LIN {X 0,Y 101.86,Z 670.766,A -85,B 0,C 180,E1 -28292.306,E2 -28292.306} C_VEL
LIN {X 0,Y 95.188,Z 678.477,A -85,B 0,C 180,E1 -28295.693,E2 -28295.693} C_VEL
LIN {X 0,Y 87.721,Z 685.98,A -85,B 0,C 180,E1 -28300.438,E2 -28300.438} C_VEL
LIN {X 0,Y 80.748,Z 692,A -85,B 0,C 180,E1 -28305.87,E2 -28305.87} C_VEL
LIN {X 0,Y 74.603,Z 696.757,A -85,B 0,C 180,E1 -28312.242,E2 -28312.242} C_VEL
LIN {X 0,Y 69.596,Z 700.393,A -85,B 0,C 180,E1 -28319.675,E2 -28319.675} C_VEL
LIN {X 0,Y 66.959,Z 702.265,A -85,B 0,C 180,E1 -28325.176,E2 -28325.176} C_VEL
LIN {X 0,Y 64.891,Z 703.687,A -85,B 0,C 180,E1 -28331.04,E2 -28331.04} C_VEL
LIN {X 0,Y 63.469,Z 704.685,A -85,B 0,C 180,E1 -28337.206,E2 -28337.206} C_VEL
LIN {X 0,Y 62.687,Z 705.298,A -85,B 0,C 180,E1 -28343.564,E2 -28343.564} C_VEL
LIN {X 0,Y 62.554,Z 705.526,A -85,B 0,C 180,E1 -28350.001,E2 -28350.001} C_VEL
LIN {X 0,Y 62.682,Z 705.324,A -85,B 0,C 180,E1 -28356.439,E2 -28356.439} C_VEL
LIN {X 0,Y 63.445,Z 704.728,A -85,B 0,C 180,E1 -28362.801,E2 -28362.801} C_VEL
LIN {X 0,Y 64.821,Z 703.747,A -85,B 0,C 180,E1 -28368.983,E2 -28368.983} C_VEL
LIN {X 0,Y 66.882,Z 702.358,A -85,B 0,C 180,E1 -28374.856,E2 -28374.856} C_VEL
LIN {X 0,Y 71.032,Z 699.448,A -85,B 0,C 180,E1 -28382.97,E2 -28382.97} C_VEL
LIN {X 0,Y 76.493,Z 695.492,A -85,B 0,C 180,E1 -28390.028,E2 -28390.028} C_VEL
LIN {X 0,Y 82.906,Z 690.364,A -85,B 0,C 180,E1 -28396.102,E2 -28396.102} C_VEL
LIN {X 0,Y 90.621,Z 683.358,A -85,B 0,C 180,E1 -28401.652,E2 -28401.652} C_VEL
LIN {X 0,Y 97.748,Z 675.871,A -85,B 0,C 180,E1 -28405.777,E2 -28405.777} C_VEL
LIN {X 0,Y 104.595,Z 667.648,A -85,B 0,C 180,E1 -28408.95,E2 -28408.95} C_VEL
LIN {X 0,Y 111.753,Z 657.491,A -85,B 0,C 180,E1 -28411.697,E2 -28411.697} C_VEL
LIN {X 0,Y 118.381,Z 646.062,A -85,B 0,C 180,E1 -28413.89,E2 -28413.89} C_VEL
LIN {X 0,Y 123.615,Z 634.711,A -85,B 0,C 180,E1 -28415.461,E2 -28415.461} C_VEL
LIN {X 0,Y 128.197,Z 621.782,A -85,B 0,C 180,E1 -28416.675,E2 -28416.675} C_VEL
LIN {X 0,Y 131.423,Z 608.945,A -85,B 0,C 180,E1 -28417.489,E2 -28417.489} C_VEL
LIN {X 0,Y 133.473,Z 595.213,A -85,B 0,C 180,E1 -28418.011,E2 -28418.011} C_VEL
LIN {X 0,Y 138.268,Z 548.092,A -85,B 0,C 180,E1 -28419.546,E2 -28419.546} C_VEL
LIN {X 0,Y 138.309,Z 545.503,A -85,B 0,C 180,E1 -28419.878,E2 -28419.878} C_VEL
LIN {X 0,Y 136.481,Z 538.988,A -85,B 0,C 180,E1 -28423.201,E2 -28423.201} C_VEL
LIN {X 0,Y 135.049,Z 534.594,A -85,B 0,C 180,E1 -28426.265,E2 -28426.265} C_VEL
LIN {X 0,Y 134.032,Z 531.605,A -85,B 0,C 180,E1 -28428.947,E2 -28428.947} C_VEL
LIN {X 0,Y 132.897,Z 528.182,A -85,B 0,C 180,E1 -28433.166,E2 -28433.166} C_VEL
LIN {X 0,Y 132.282,Z 525.748,A -85,B 0,C 180,E1 -28438.478,E2 -28438.478} C_VEL
LIN {X 0,Y 132.299,Z 525.196,A -85,B 0,C 180,E1 -28440,E2 -28440} C_VEL
LIN {X 0,Y 132.523,Z 525.208,A -85,B 0,C 180,E1 -28443.42,E2 -28443.42} C_VEL
LIN {X 0,Y 133.793,Z 527.549,A -85,B 0,C 180,E1 -28449.448,E2 -28449.448} C_VEL
LIN {X 0,Y 135.294,Z 530.109,A -85,B 0,C 180,E1 -28453.327,E2 -28453.327} C_VEL
LIN {X 0,Y 137.511,Z 534.497,A -85,B 0,C 180,E1 -28457.569,E2 -28457.569} C_VEL
LIN {X 0,Y 138.613,Z 536.926,A -85,B 0,C 180,E1 -28459.339,E2 -28459.339} C_VEL
LIN {X 0,Y 137.874,Z 550.601,A -85,B 0,C 180,E1 -28460.537,E2 -28460.537} C_VEL
LIN {X 0,Y 132.225,Z 603.924,A -85,B 0,C 180,E1 -28462.263,E2 -28462.263} C_VEL
LIN {X 0,Y 129.662,Z 616.387,A -85,B 0,C 180,E1 -28462.86,E2 -28462.86} C_VEL
LIN {X 0,Y 125.786,Z 629.073,A -85,B 0,C 180,E1 -28463.805,E2 -28463.805} C_VEL
LIN {X 0,Y 121.232,Z 640.398,A -85,B 0,C 180,E1 -28465.066,E2 -28465.066} C_VEL
LIN {X 0,Y 115.246,Z 652.046,A -85,B 0,C 180,E1 -28466.889,E2 -28466.889} C_VEL
LIN {X 0,Y 108.673,Z 662.454,A -85,B 0,C 180,E1 -28469.182,E2 -28469.182} C_VEL
LIN {X 0,Y 101.589,Z 671.843,A -85,B 0,C 180,E1 -28472.062,E2 -28472.062} C_VEL
LIN {X 0,Y 93.505,Z 680.856,A -85,B 0,C 180,E1 -28476.099,E2 -28476.099} C_VEL
LIN {X 0,Y 85.896,Z 688.299,A -85,B 0,C 180,E1 -28481.118,E2 -28481.118} C_VEL
LIN {X 0,Y 80.359,Z 693.02,A -85,B 0,C 180,E1 -28485.599,E2 -28485.599} C_VEL
LIN {X 0,Y 74.261,Z 697.769,A -85,B 0,C 180,E1 -28492.036,E2 -28492.036} C_VEL
LIN {X 0,Y 69.197,Z 701.394,A -85,B 0,C 180,E1 -28499.48,E2 -28499.48} C_VEL
LIN {X 0,Y 66.631,Z 703.263,A -85,B 0,C 180,E1 -28505.044,E2 -28505.044} C_VEL
LIN {X 0,Y 64.645,Z 704.669,A -85,B 0,C 180,E1 -28510.964,E2 -28510.964} C_VEL
LIN {X 0,Y 63.349,Z 705.663,A -85,B 0,C 180,E1 -28517.179,E2 -28517.179} C_VEL
LIN {X 0,Y 62.666,Z 706.269,A -85,B 0,C 180,E1 -28523.56,E2 -28523.56} C_VEL
LIN {X 0,Y 62.617,Z 706.48,A -85,B 0,C 180,E1 -28529.999,E2 -28529.999} C_VEL
LIN {X 0,Y 62.666,Z 706.25,A -85,B 0,C 180,E1 -28536.438,E2 -28536.438} C_VEL
LIN {X 0,Y 63.349,Z 705.631,A -85,B 0,C 180,E1 -28542.819,E2 -28542.819} C_VEL
LIN {X 0,Y 64.645,Z 704.625,A -85,B 0,C 180,E1 -28549.034,E2 -28549.034} C_VEL
LIN {X 0,Y 66.632,Z 703.194,A -85,B 0,C 180,E1 -28554.954,E2 -28554.954} C_VEL
LIN {X 0,Y 70.759,Z 700.231,A -85,B 0,C 180,E1 -28563.111,E2 -28563.111} C_VEL
LIN {X 0,Y 76.222,Z 696.212,A -85,B 0,C 180,E1 -28570.197,E2 -28570.197} C_VEL
LIN {X 0,Y 82.628,Z 691.019,A -85,B 0,C 180,E1 -28576.3,E2 -28576.3} C_VEL
LIN {X 0,Y 89.725,Z 684.486,A -85,B 0,C 180,E1 -28581.561,E2 -28581.561} C_VEL
LIN {X 0,Y 97.461,Z 676.359,A -85,B 0,C 180,E1 -28586.023,E2 -28586.023} C_VEL
LIN {X 0,Y 104.564,Z 667.747,A -85,B 0,C 180,E1 -28589.248,E2 -28589.248} C_VEL
LIN {X 0,Y 104.524,Z 666.501,A -85,B 0,C 180,E1 -28590.516,E2 -28590.516} C_VEL
LIN {X 0,Y 98.912,Z 662.815,A -85,B 0,C 180,E1 -28602.135,E2 -28602.135} C_VEL
LIN {X 0,Y 98.359,Z 659.574,A -85,B 0,C 180,E1 -28609.71,E2 -28609.71} C_VEL
LIN {X 0,Y 99.161,Z 657.199,A -85,B 0,C 180,E1 -28613.724,E2 -28613.724} C_VEL
LIN {X 0,Y 99.935,Z 655.554,A -85,B 0,C 180,E1 -28616.976,E2 -28616.976} C_VEL
LIN {X 0,Y 102.399,Z 652.842,A -85,B 0,C 180,E1 -28626.921,E2 -28626.921} C_VEL
LIN {X 0,Y 104.174,Z 651.421,A -85,B 0,C 180,E1 -28629.967,E2 -28629.967} C_VEL
LIN {X 0,Y 104.937,Z 650.77,A -85,B 0,C 180,E1 -28630.903,E2 -28630.903} C_VEL
LIN {X 0,Y 109.265,Z 646.893,A -85,B 0,C 180,E1 -28635.098,E2 -28635.098} C_VEL
LIN {X 0,Y 116.042,Z 640.504,A -85,B 0,C 180,E1 -28639.805,E2 -28639.805} C_VEL
LIN {X 0,Y 119.153,Z 637.397,A -85,B 0,C 180,E1 -28641.632,E2 -28641.632} C_VEL
LIN {X 0,Y 118.879,Z 638.512,A -85,B 0,C 180,E1 -28642.044,E2 -28642.044} C_VEL
LIN {X 0,Y 113.178,Z 649.684,A -85,B 0,C 180,E1 -28643.662,E2 -28643.662} C_VEL
LIN {X 0,Y 106.362,Z 660.356,A -85,B 0,C 180,E1 -28645.805,E2 -28645.805} C_VEL
LIN {X 0,Y 98.252,Z 670.818,A -85,B 0,C 180,E1 -28648.808,E2 -28648.808} C_VEL
LIN {X 0,Y 91.212,Z 678.529,A -85,B 0,C 180,E1 -28652.053,E2 -28652.053} C_VEL
LIN {X 0,Y 83.223,Z 686.089,A -85,B 0,C 180,E1 -28656.757,E2 -28656.757} C_VEL
LIN {X 0,Y 75.792,Z 692.054,A -85,B 0,C 180,E1 -28662.114,E2 -28662.114} C_VEL
LIN {X 0,Y 69.122,Z 696.812,A -85,B 0,C 180,E1 -28668.633,E2 -28668.633} C_VEL
LIN {X 0,Y 63.538,Z 700.448,A -85,B 0,C 180,E1 -28676.424,E2 -28676.424} C_VEL
LIN {X 0,Y 60.561,Z 702.319,A -85,B 0,C 180,E1 -28682.343,E2 -28682.343} C_VEL
LIN {X 0,Y 58.212,Z 703.741,A -85,B 0,C 180,E1 -28688.766,E2 -28688.766} C_VEL
LIN {X 0,Y 55.63,Z 705.352,A -85,B 0,C 180,E1 -28702.743,E2 -28702.743} C_VEL
LIN {X 0,Y 55.473,Z 705.58,A -85,B 0,C 180,E1 -28710.001,E2 -28710.001} C_VEL
LIN {X 0,Y 55.626,Z 705.378,A -85,B 0,C 180,E1 -28717.259,E2 -28717.259} C_VEL
LIN {X 0,Y 56.529,Z 704.781,A -85,B 0,C 180,E1 -28724.399,E2 -28724.399} C_VEL
LIN {X 0,Y 58.15,Z 703.8,A -85,B 0,C 180,E1 -28731.26,E2 -28731.26} C_VEL
LIN {X 0,Y 60.49,Z 702.411,A -85,B 0,C 180,E1 -28737.695,E2 -28737.695} C_VEL
LIN {X 0,Y 65.174,Z 699.501,A -85,B 0,C 180,E1 -28746.378,E2 -28746.378} C_VEL
LIN {X 0,Y 71.197,Z 695.544,A -85,B 0,C 180,E1 -28753.709,E2 -28753.709} C_VEL
LIN {X 0,Y 78.142,Z 690.415,A -85,B 0,C 180,E1 -28759.862,E2 -28759.862} C_VEL
LIN {X 0,Y 85.789,Z 683.952,A -85,B 0,C 180,E1 -28765.008,E2 -28765.008} C_VEL
LIN {X 0,Y 93.93,Z 675.919,A -85,B 0,C 180,E1 -28769.368,E2 -28769.368} C_VEL
LIN {X 0,Y 101.109,Z 667.693,A -85,B 0,C 180,E1 -28772.407,E2 -28772.407} C_VEL
LIN {X 0,Y 108.564,Z 657.532,A -85,B 0,C 180,E1 -28775.001,E2 -28775.001} C_VEL
LIN {X 0,Y 115.434,Z 646.099,A -85,B 0,C 180,E1 -28777.054,E2 -28777.054} C_VEL
LIN {X 0,Y 120.841,Z 634.739,A -85,B 0,C 180,E1 -28778.522,E2 -28778.522} C_VEL
LIN {X 0,Y 125.558,Z 621.799,A -85,B 0,C 180,E1 -28779.649,E2 -28779.649} C_VEL
LIN {X 0,Y 128.829,Z 609.172,A -85,B 0,C 180,E1 -28780.39,E2 -28780.39} C_VEL
LIN {X 0,Y 130.949,Z 595.406,A -85,B 0,C 180,E1 -28780.886,E2 -28780.886} C_VEL
LIN {X 0,Y 135.81,Z 549.367,A -85,B 0,C 180,E1 -28782.304,E2 -28782.304} C_VEL
LIN {X 0,Y 134.47,Z 544.016,A -85,B 0,C 180,E1 -28785.239,E2 -28785.239} C_VEL
LIN {X 0,Y 132.962,Z 538.749,A -85,B 0,C 180,E1 -28789.339,E2 -28789.339} C_VEL
LIN {X 0,Y 131.864,Z 535.005,A -85,B 0,C 180,E1 -28793.881,E2 -28793.881} C_VEL
LIN {X 0,Y 131.402,Z 532.741,A -85,B 0,C 180,E1 -28798.851,E2 -28798.851} C_VEL
LIN {X 0,Y 131.424,Z 532.32,A -85,B 0,C 180,E1 -28800,E2 -28800} C_VEL
LIN {X 0,Y 131.67,Z 532.377,A -85,B 0,C 180,E1 -28803.634,E2 -28803.634} C_VEL
LIN {X 0,Y 132.86,Z 534.677,A -85,B 0,C 180,E1 -28809.323,E2 -28809.323} C_VEL
LIN {X 0,Y 134.08,Z 536.98,A -85,B 0,C 180,E1 -28812.679,E2 -28812.679} C_VEL
LIN {X 0,Y 135.868,Z 540.882,A -85,B 0,C 180,E1 -28816.432,E2 -28816.432} C_VEL
LIN {X 0,Y 136.117,Z 541.431,A -85,B 0,C 180,E1 -28816.884,E2 -28816.884} C_VEL
LIN {X 0,Y 135.492,Z 551.207,A -85,B 0,C 180,E1 -28817.742,E2 -28817.742} C_VEL
LIN {X 0,Y 129.707,Z 603.961,A -85,B 0,C 180,E1 -28819.366,E2 -28819.366} C_VEL
LIN {X 0,Y 126.879,Z 617.11,A -85,B 0,C 180,E1 -28819.96,E2 -28819.96} C_VEL
LIN {X 0,Y 122.703,Z 630.146,A -85,B 0,C 180,E1 -28820.879,E2 -28820.879} C_VEL
LIN {X 0,Y 117.624,Z 641.987,A -85,B 0,C 180,E1 -28822.159,E2 -28822.159} C_VEL
LIN {X 0,Y 111.461,Z 653.275,A -85,B 0,C 180,E1 -28823.895,E2 -28823.895} C_VEL
LIN {X 0,Y 104.642,Z 663.464,A -85,B 0,C 180,E1 -28826.063,E2 -28826.063} C_VEL
LIN {X 0,Y 97.991,Z 671.797,A -85,B 0,C 180,E1 -28828.526,E2 -28828.526} C_VEL
LIN {X 0,Y 89.498,Z 680.808,A -85,B 0,C 180,E1 -28832.416,E2 -28832.416} C_VEL
LIN {X 0,Y 82.031,Z 687.662,A -85,B 0,C 180,E1 -28836.85,E2 -28836.85} C_VEL
LIN {X 0,Y 75.449,Z 692.969,A -85,B 0,C 180,E1 -28841.823,E2 -28841.823} C_VEL
LIN {X 0,Y 68.79,Z 697.717,A -85,B 0,C 180,E1 -28848.387,E2 -28848.387} C_VEL
LIN {X 0,Y 63.157,Z 701.341,A -85,B 0,C 180,E1 -28856.192,E2 -28856.192} C_VEL
LIN {X 0,Y 60.238,Z 703.21,A -85,B 0,C 180,E1 -28862.18,E2 -28862.18} C_VEL
LIN {X 0,Y 57.959,Z 704.615,A -85,B 0,C 180,E1 -28868.667,E2 -28868.667} C_VEL
LIN {X 0,Y 56.418,Z 705.609,A -85,B 0,C 180,E1 -28875.572,E2 -28875.572} C_VEL
LIN {X 0,Y 55.608,Z 706.215,A -85,B 0,C 180,E1 -28882.738,E2 -28882.738} C_VEL
LIN {X 0,Y 55.518,Z 706.426,A -85,B 0,C 180,E1 -28889.999,E2 -28889.999} C_VEL
LIN {X 0,Y 55.608,Z 706.196,A -85,B 0,C 180,E1 -28897.26,E2 -28897.26} C_VEL
LIN {X 0,Y 56.44,Z 705.577,A -85,B 0,C 180,E1 -28904.42,E2 -28904.42} C_VEL
LIN {X 0,Y 57.959,Z 704.57,A -85,B 0,C 180,E1 -28911.331,E2 -28911.331} C_VEL
LIN {X 0,Y 60.24,Z 703.139,A -85,B 0,C 180,E1 -28917.817,E2 -28917.817} C_VEL
LIN {X 0,Y 64.909,Z 700.176,A -85,B 0,C 180,E1 -28926.548,E2 -28926.548} C_VEL
LIN {X 0,Y 70.917,Z 696.158,A -85,B 0,C 180,E1 -28933.924,E2 -28933.924} C_VEL
LIN {X 0,Y 77.887,Z 690.966,A -85,B 0,C 180,E1 -28940.083,E2 -28940.083} C_VEL
LIN {X 0,Y 85.468,Z 684.432,A -85,B 0,C 180,E1 -28945.315,E2 -28945.315} C_VEL
LIN {X 0,Y 93.674,Z 676.307,A -85,B 0,C 180,E1 -28949.632,E2 -28949.632} C_VEL
LIN {X 0,Y 98.134,Z 671.326,A -85,B 0,C 180,E1 -28951.527,E2 -28951.527} C_VEL
LIN {X 0,Y 97.705,Z 670.632,A -85,B 0,C 180,E1 -28952.853,E2 -28952.853} C_VEL
LIN {X 0,Y 93.931,Z 667.818,A -85,B 0,C 180,E1 -28962.586,E2 -28962.586} C_VEL
LIN {X 0,Y 93.807,Z 664.313,A -85,B 0,C 180,E1 -28971.383,E2 -28971.383} C_VEL
LIN {X 0,Y 97.057,Z 659.101,A -85,B 0,C 180,E1 -28980,E2 -28980} C_VEL
LIN {X 0,Y 101.182,Z 654.304,A -85,B 0,C 180,E1 -28985.981,E2 -28985.981} C_VEL
LIN {X 0,Y 104.937,Z 650.77,A -85,B 0,C 180,E1 -28990.903,E2 -28990.903} C_VEL
LIN {X 0,Y 105.764,Z 650.311,A -85,B 0,C 180,E1 -28992.232,E2 -28992.232} C_VEL
LIN {X 0,Y 106.24,Z 650.817,A -85,B 0,C 180,E1 -28994.121,E2 -28994.121} C_VEL
LIN {X 0,Y 106.094,Z 652.648,A -85,B 0,C 180,E1 -28996.445,E2 -28996.445} C_VEL
LIN {X 0,Y 104.964,Z 656.019,A -85,B 0,C 180,E1 -28999.009,E2 -28999.009} C_VEL
LIN {X 0,Y 102.937,Z 660.296,A -85,B 0,C 180,E1 -29001.374,E2 -29001.374} C_VEL
LIN {X 0,Y 100.077,Z 664.814,A -85,B 0,C 180,E1 -29003.248,E2 -29003.248} C_VEL
LIN {X 0,Y 98.91,Z 666.324,A -85,B 0,C 180,E1 -29003.721,E2 -29003.721} C_VEL
LIN {X 0,Y 90.56,Z 675.661,A -85,B 0,C 180,E1 -29006.815,E2 -29006.815} C_VEL
LIN {X 0,Y 81.98,Z 683.754,A -85,B 0,C 180,E1 -29010.988,E2 -29010.988} C_VEL
LIN {X 0,Y 73.799,Z 690.26,A -85,B 0,C 180,E1 -29015.956,E2 -29015.956} C_VEL
LIN {X 0,Y 66.289,Z 695.43,A -85,B 0,C 180,E1 -29022.086,E2 -29022.086} C_VEL
LIN {X 0,Y 59.657,Z 699.429,A -85,B 0,C 180,E1 -29029.615,E2 -29029.615} C_VEL
LIN {X 0,Y 54.351,Z 702.374,A -85,B 0,C 180,E1 -29038.854,E2 -29038.854} C_VEL
LIN {X 0,Y 51.655,Z 703.796,A -85,B 0,C 180,E1 -29045.911,E2 -29045.911} C_VEL
LIN {X 0,Y 48.602,Z 705.406,A -85,B 0,C 180,E1 -29061.687,E2 -29061.687} C_VEL
LIN {X 0,Y 48.375,Z 705.634,A -85,B 0,C 180,E1 -29070.001,E2 -29070.001} C_VEL
LIN {X 0,Y 48.597,Z 705.431,A -85,B 0,C 180,E1 -29078.316,E2 -29078.316} C_VEL
LIN {X 0,Y 49.682,Z 704.835,A -85,B 0,C 180,E1 -29086.436,E2 -29086.436} C_VEL
LIN {X 0,Y 51.586,Z 703.854,A -85,B 0,C 180,E1 -29094.125,E2 -29094.125} C_VEL
LIN {X 0,Y 54.287,Z 702.465,A -85,B 0,C 180,E1 -29101.189,E2 -29101.189} C_VEL
LIN {X 0,Y 59.599,Z 699.553,A -85,B 0,C 180,E1 -29110.436,E2 -29110.436} C_VEL
LIN {X 0,Y 66.244,Z 695.595,A -85,B 0,C 180,E1 -29117.959,E2 -29117.959} C_VEL
LIN {X 0,Y 73.763,Z 690.465,A -85,B 0,C 180,E1 -29124.085,E2 -29124.085} C_VEL
LIN {X 0,Y 81.917,Z 684.001,A -85,B 0,C 180,E1 -29129.089,E2 -29129.089} C_VEL
LIN {X 0,Y 90.503,Z 675.966,A -85,B 0,C 180,E1 -29133.259,E2 -29133.259} C_VEL
LIN {X 0,Y 98.016,Z 667.739,A -85,B 0,C 180,E1 -29136.095,E2 -29136.095} C_VEL
LIN {X 0,Y 105.758,Z 657.574,A -85,B 0,C 180,E1 -29138.492,E2 -29138.492} C_VEL
LIN {X 0,Y 112.858,Z 646.135,A -85,B 0,C 180,E1 -29140.372,E2 -29140.372} C_VEL
LIN {X 0,Y 118.427,Z 634.767,A -85,B 0,C 180,E1 -29141.719,E2 -29141.719} C_VEL
LIN {X 0,Y 123.273,Z 621.816,A -85,B 0,C 180,E1 -29142.739,E2 -29142.739} C_VEL
LIN {X 0,Y 126.542,Z 609.541,A -85,B 0,C 180,E1 -29143.401,E2 -29143.401} C_VEL
LIN {X 0,Y 128.842,Z 595.013,A -85,B 0,C 180,E1 -29143.869,E2 -29143.869} C_VEL
LIN {X 0,Y 133.449,Z 552.752,A -85,B 0,C 180,E1 -29145.095,E2 -29145.095} C_VEL
LIN {X 0,Y 132.365,Z 548.001,A -85,B 0,C 180,E1 -29148.127,E2 -29148.127} C_VEL
LIN {X 0,Y 131.551,Z 544.776,A -85,B 0,C 180,E1 -29150.971,E2 -29150.971} C_VEL
LIN {X 0,Y 130.816,Z 541.688,A -85,B 0,C 180,E1 -29154.85,E2 -29154.85} C_VEL
LIN {X 0,Y 130.535,Z 539.591,A -85,B 0,C 180,E1 -29159.614,E2 -29159.614} C_VEL
LIN {X 0,Y 130.77,Z 539.401,A -85,B 0,C 180,E1 -29163.37,E2 -29163.37} C_VEL
LIN {X 0,Y 131.817,Z 541.585,A -85,B 0,C 180,E1 -29168.817,E2 -29168.817} C_VEL
LIN {X 0,Y 132.81,Z 543.717,A -85,B 0,C 180,E1 -29171.833,E2 -29171.833} C_VEL
LIN {X 0,Y 133.861,Z 546.095,A -85,B 0,C 180,E1 -29174.345,E2 -29174.345} C_VEL
LIN {X 0,Y 133.37,Z 552.487,A -85,B 0,C 180,E1 -29174.875,E2 -29174.875} C_VEL
LIN {X 0,Y 127.418,Z 604.64,A -85,B 0,C 180,E1 -29176.368,E2 -29176.368} C_VEL
LIN {X 0,Y 124.44,Z 617.833,A -85,B 0,C 180,E1 -29176.943,E2 -29176.943} C_VEL
LIN {X 0,Y 120.358,Z 630.122,A -85,B 0,C 180,E1 -29177.722,E2 -29177.722} C_VEL
LIN {X 0,Y 115.137,Z 641.953,A -85,B 0,C 180,E1 -29178.89,E2 -29178.89} C_VEL
LIN {X 0,Y 108.777,Z 653.236,A -85,B 0,C 180,E1 -29180.471,E2 -29180.471} C_VEL
LIN {X 0,Y 101.723,Z 663.42,A -85,B 0,C 180,E1 -29182.469,E2 -29182.469} C_VEL
LIN {X 0,Y 94.796,Z 671.751,A -85,B 0,C 180,E1 -29184.741,E2 -29184.741} C_VEL
LIN {X 0,Y 85.886,Z 680.76,A -85,B 0,C 180,E1 -29188.396,E2 -29188.396} C_VEL
LIN {X 0,Y 77.34,Z 688.121,A -85,B 0,C 180,E1 -29193.04,E2 -29193.04} C_VEL
LIN {X 0,Y 70.913,Z 692.918,A -85,B 0,C 180,E1 -29197.545,E2 -29197.545} C_VEL
LIN {X 0,Y 63.644,Z 697.665,A -85,B 0,C 180,E1 -29204.127,E2 -29204.127} C_VEL
LIN {X 0,Y 57.369,Z 701.288,A -85,B 0,C 180,E1 -29212.226,E2 -29212.226} C_VEL
LIN {X 0,Y 54.038,Z 703.157,A -85,B 0,C 180,E1 -29218.651,E2 -29218.651} C_VEL
LIN {X 0,Y 51.397,Z 704.561,A -85,B 0,C 180,E1 -29225.78,E2 -29225.78} C_VEL
LIN {X 0,Y 48.577,Z 706.161,A -85,B 0,C 180,E1 -29241.68,E2 -29241.68} C_VEL
LIN {X 0,Y 48.436,Z 706.372,A -85,B 0,C 180,E1 -29249.999,E2 -29249.999} C_VEL
LIN {X 0,Y 48.579,Z 706.141,A -85,B 0,C 180,E1 -29258.317,E2 -29258.317} C_VEL
LIN {X 0,Y 49.573,Z 705.522,A -85,B 0,C 180,E1 -29266.471,E2 -29266.471} C_VEL
LIN {X 0,Y 51.397,Z 704.516,A -85,B 0,C 180,E1 -29274.217,E2 -29274.217} C_VEL
LIN {X 0,Y 54.04,Z 703.084,A -85,B 0,C 180,E1 -29281.345,E2 -29281.345} C_VEL
LIN {X 0,Y 59.341,Z 700.122,A -85,B 0,C 180,E1 -29290.646,E2 -29290.646} C_VEL
LIN {X 0,Y 65.96,Z 696.104,A -85,B 0,C 180,E1 -29298.231,E2 -29298.231} C_VEL
LIN {X 0,Y 73.516,Z 690.912,A -85,B 0,C 180,E1 -29304.348,E2 -29304.348} C_VEL
LIN {X 0,Y 81.621,Z 684.379,A -85,B 0,C 180,E1 -29309.435,E2 -29309.435} C_VEL
LIN {X 0,Y 90.286,Z 676.255,A -85,B 0,C 180,E1 -29313.531,E2 -29313.531} C_VEL
LIN {X 0,Y 91.323,Z 674.766,A -85,B 0,C 180,E1 -29314.607,E2 -29314.607} C_VEL
LIN {X 0,Y 88.963,Z 672.945,A -85,B 0,C 180,E1 -29321.579,E2 -29321.579} C_VEL
LIN {X 0,Y 88.686,Z 669.789,A -85,B 0,C 180,E1 -29330.881,E2 -29330.881} C_VEL
LIN {X 0,Y 89.847,Z 667.724,A -85,B 0,C 180,E1 -29335.514,E2 -29335.514} C_VEL
LIN {X 0,Y 93.347,Z 663.616,A -85,B 0,C 180,E1 -29342.422,E2 -29342.422} C_VEL
LIN {X 0,Y 97.915,Z 659.201,A -85,B 0,C 180,E1 -29348.254,E2 -29348.254} C_VEL
LIN {X 0,Y 104.701,Z 653.863,A -85,B 0,C 180,E1 -29355.575,E2 -29355.575} C_VEL
LIN {X 0,Y 110.24,Z 649.405,A -85,B 0,C 180,E1 -29359.567,E2 -29359.567} C_VEL
LIN {X 0,Y 109.931,Z 650.703,A -85,B 0,C 180,E1 -29360.443,E2 -29360.443} C_VEL
LIN {X 0,Y 102.69,Z 661.452,A -85,B 0,C 180,E1 -29362.494,E2 -29362.494} C_VEL
LIN {X 0,Y 98.91,Z 666.324,A -85,B 0,C 180,E1 -29363.721,E2 -29363.721} C_VEL
LIN {X 0,Y 95.093,Z 670.569,A -85,B 0,C 180,E1 -29364.625,E2 -29364.625} C_VEL
LIN {X 0,Y 87.709,Z 677.086,A -85,B 0,C 180,E1 -29365.376,E2 -29365.376} C_VEL
LIN {X 0,Y 79.911,Z 682.975,A -85,B 0,C 180,E1 -29366.473,E2 -29366.473} C_VEL
LIN {X 0,Y 75.514,Z 686.232,A -85,B 0,C 180,E1 -29368.092,E2 -29368.092} C_VEL
LIN {X 0,Y 67.07,Z 692.161,A -85,B 0,C 180,E1 -29373.042,E2 -29373.042} C_VEL
LIN {X 0,Y 59.211,Z 696.92,A -85,B 0,C 180,E1 -29379.511,E2 -29379.511} C_VEL
LIN {X 0,Y 52.251,Z 700.557,A -85,B 0,C 180,E1 -29387.739,E2 -29387.739} C_VEL
LIN {X 0,Y 48.399,Z 702.428,A -85,B 0,C 180,E1 -29394.492,E2 -29394.492} C_VEL
LIN {X 0,Y 45.242,Z 703.85,A -85,B 0,C 180,E1 -29402.225,E2 -29402.225} C_VEL
LIN {X 0,Y 41.586,Z 705.461,A -85,B 0,C 180,E1 -29420.272,E2 -29420.272} C_VEL
LIN {X 0,Y 41.293,Z 705.688,A -85,B 0,C 180,E1 -29430.001,E2 -29430.001} C_VEL
LIN {X 0,Y 41.581,Z 705.485,A -85,B 0,C 180,E1 -29439.732,E2 -29439.732} C_VEL
LIN {X 0,Y 42.903,Z 704.889,A -85,B 0,C 180,E1 -29449.126,E2 -29449.126} C_VEL
LIN {X 0,Y 45.182,Z 703.907,A -85,B 0,C 180,E1 -29457.818,E2 -29457.818} C_VEL
LIN {X 0,Y 48.342,Z 702.518,A -85,B 0,C 180,E1 -29465.559,E2 -29465.559} C_VEL
LIN {X 0,Y 54.387,Z 699.606,A -85,B 0,C 180,E1 -29475.295,E2 -29475.295} C_VEL
LIN {X 0,Y 61.715,Z 695.647,A -85,B 0,C 180,E1 -29482.861,E2 -29482.861} C_VEL
LIN {X 0,Y 69.835,Z 690.516,A -85,B 0,C 180,E1 -29488.808,E2 -29488.808} C_VEL
LIN {X 0,Y 78.503,Z 684.05,A -85,B 0,C 180,E1 -29493.543,E2 -29493.543} C_VEL
LIN {X 0,Y 87.535,Z 676.014,A -85,B 0,C 180,E1 -29497.417,E2 -29497.417} C_VEL
LIN {X 0,Y 95.358,Z 667.784,A -85,B 0,C 180,E1 -29500.002,E2 -29500.002} C_VEL
LIN {X 0,Y 103.365,Z 657.615,A -85,B 0,C 180,E1 -29502.157,E2 -29502.157} C_VEL
LIN {X 0,Y 110.677,Z 646.172,A -85,B 0,C 180,E1 -29503.833,E2 -29503.833} C_VEL
LIN {X 0,Y 116.399,Z 634.795,A -85,B 0,C 180,E1 -29505.033,E2 -29505.033} C_VEL
LIN {X 0,Y 121.361,Z 621.831,A -85,B 0,C 180,E1 -29505.93,E2 -29505.93} C_VEL
LIN {X 0,Y 124.869,Z 608.767,A -85,B 0,C 180,E1 -29506.537,E2 -29506.537} C_VEL
LIN {X 0,Y 127.15,Z 594.103,A -85,B 0,C 180,E1 -29506.962,E2 -29506.962} C_VEL
LIN {X 0,Y 131.378,Z 556.367,A -85,B 0,C 180,E1 -29507.996,E2 -29507.996} C_VEL
LIN {X 0,Y 130.491,Z 551.836,A -85,B 0,C 180,E1 -29511.482,E2 -29511.482} C_VEL
LIN {X 0,Y 129.832,Z 548.516,A -85,B 0,C 180,E1 -29515.589,E2 -29515.589} C_VEL
LIN {X 0,Y 129.671,Z 546.588,A -85,B 0,C 180,E1 -29520,E2 -29520} C_VEL
LIN {X 0,Y 129.926,Z 546.605,A -85,B 0,C 180,E1 -29523.683,E2 -29523.683} C_VEL
LIN {X 0,Y 130.936,Z 548.842,A -85,B 0,C 180,E1 -29528.877,E2 -29528.877} C_VEL
LIN {X 0,Y 131.844,Z 551.233,A -85,B 0,C 180,E1 -29531.785,E2 -29531.785} C_VEL
LIN {X 0,Y 125.803,Z 603.462,A -85,B 0,C 180,E1 -29533.235,E2 -29533.235} C_VEL
LIN {X 0,Y 122.97,Z 616.366,A -85,B 0,C 180,E1 -29533.688,E2 -29533.688} C_VEL
LIN {X 0,Y 118.808,Z 629.008,A -85,B 0,C 180,E1 -29534.382,E2 -29534.382} C_VEL
LIN {X 0,Y 113.863,Z 640.303,A -85,B 0,C 180,E1 -29535.325,E2 -29535.325} C_VEL
LIN {X 0,Y 107.308,Z 651.93,A -85,B 0,C 180,E1 -29536.692,E2 -29536.692} C_VEL
LIN {X 0,Y 100.026,Z 662.326,A -85,B 0,C 180,E1 -29538.459,E2 -29538.459} C_VEL
LIN {X 0,Y 92.049,Z 671.705,A -85,B 0,C 180,E1 -29540.722,E2 -29540.722} C_VEL
LIN {X 0,Y 82.742,Z 680.711,A -85,B 0,C 180,E1 -29544.061,E2 -29544.061} C_VEL
LIN {X 0,Y 73.05,Z 688.566,A -85,B 0,C 180,E1 -29548.753,E2 -29548.753} C_VEL
LIN {X 0,Y 64.069,Z 694.589,A -85,B 0,C 180,E1 -29554.641,E2 -29554.641} C_VEL
LIN {X 0,Y 56.459,Z 698.942,A -85,B 0,C 180,E1 -29561.677,E2 -29561.677} C_VEL
LIN {X 0,Y 51.923,Z 701.236,A -85,B 0,C 180,E1 -29567.406,E2 -29567.406} C_VEL
LIN {X 0,Y 48.082,Z 703.103,A -85,B 0,C 180,E1 -29574.218,E2 -29574.218} C_VEL
LIN {X 0,Y 44.995,Z 704.508,A -85,B 0,C 180,E1 -29582.056,E2 -29582.056} C_VEL
LIN {X 0,Y 42.789,Z 705.501,A -85,B 0,C 180,E1 -29590.821,E2 -29590.821} C_VEL
LIN {X 0,Y 41.558,Z 706.107,A -85,B 0,C 180,E1 -29600.262,E2 -29600.262} C_VEL
LIN {X 0,Y 41.337,Z 706.318,A -85,B 0,C 180,E1 -29609.999,E2 -29609.999} C_VEL
LIN {X 0,Y 41.56,Z 706.087,A -85,B 0,C 180,E1 -29619.735,E2 -29619.735} C_VEL
LIN {X 0,Y 42.802,Z 705.468,A -85,B 0,C 180,E1 -29629.17,E2 -29629.17} C_VEL
LIN {X 0,Y 44.995,Z 704.461,A -85,B 0,C 180,E1 -29637.941,E2 -29637.941} C_VEL
LIN {X 0,Y 48.083,Z 703.03,A -85,B 0,C 180,E1 -29645.777,E2 -29645.777} C_VEL
LIN {X 0,Y 54.14,Z 700.067,A -85,B 0,C 180,E1 -29655.557,E2 -29655.557} C_VEL
LIN {X 0,Y 61.436,Z 696.049,A -85,B 0,C 180,E1 -29663.202,E2 -29663.202} C_VEL
LIN {X 0,Y 69.603,Z 690.858,A -85,B 0,C 180,E1 -29669.122,E2 -29669.122} C_VEL
LIN {X 0,Y 78.234,Z 684.326,A -85,B 0,C 180,E1 -29673.939,E2 -29673.939} C_VEL
LIN {X 0,Y 84.263,Z 679.134,A -85,B 0,C 180,E1 -29676.558,E2 -29676.558} C_VEL
LIN {X 0,Y 83.76,Z 677.769,A -85,B 0,C 180,E1 -29680.389,E2 -29680.389} C_VEL
LIN {X 0,Y 83.311,Z 674.934,A -85,B 0,C 180,E1 -29690.287,E2 -29690.287} C_VEL
LIN {X 0,Y 84.553,Z 672.849,A -85,B 0,C 180,E1 -29695.89,E2 -29695.89} C_VEL
LIN {X 0,Y 89.178,Z 668.304,A -85,B 0,C 180,E1 -29704.52,E2 -29704.52} C_VEL
LIN {X 0,Y 94.539,Z 663.933,A -85,B 0,C 180,E1 -29710.711,E2 -29710.711} C_VEL
LIN {X 0,Y 102.07,Z 658.832,A -85,B 0,C 180,E1 -29717.959,E2 -29717.959} C_VEL
LIN {X 0,Y 101.206,Z 660.178,A -85,B 0,C 180,E1 -29718.48,E2 -29718.48} C_VEL
LIN {X 0,Y 93.836,Z 669.167,A -85,B 0,C 180,E1 -29720.576,E2 -29720.576} C_VEL
LIN {X 0,Y 86.048,Z 677.176,A -85,B 0,C 180,E1 -29723.243,E2 -29723.243} C_VEL
LIN {X 0,Y 76.538,Z 685.456,A -85,B 0,C 180,E1 -29727.552,E2 -29727.552} C_VEL
LIN {X 0,Y 75.514,Z 686.232,A -85,B 0,C 180,E1 -29728.092,E2 -29728.092} C_VEL
LIN {X 0,Y 71.049,Z 689.307,A -85,B 0,C 180,E1 -29729.965,E2 -29729.965} C_VEL
LIN {X 0,Y 62.659,Z 693.847,A -85,B 0,C 180,E1 -29732.298,E2 -29732.298} C_VEL
LIN {X 0,Y 54.096,Z 697.69,A -85,B 0,C 180,E1 -29735.499,E2 -29735.499} C_VEL
LIN {X 0,Y 49.541,Z 699.601,A -85,B 0,C 180,E1 -29739.101,E2 -29739.101} C_VEL
LIN {X 0,Y 42.809,Z 702.483,A -85,B 0,C 180,E1 -29748.954,E2 -29748.954} C_VEL
LIN {X 0,Y 39.087,Z 703.905,A -85,B 0,C 180,E1 -29757.358,E2 -29757.358} C_VEL
LIN {X 0,Y 34.598,Z 705.515,A -85,B 0,C 180,E1 -29778.281,E2 -29778.281} C_VEL
LIN {X 0,Y 34.187,Z 705.742,A -85,B 0,C 180,E1 -29790.002,E2 -29790.002} C_VEL
LIN {X 0,Y 34.593,Z 705.539,A -85,B 0,C 180,E1 -29801.724,E2 -29801.724} C_VEL
LIN {X 0,Y 36.264,Z 704.943,A -85,B 0,C 180,E1 -29812.807,E2 -29812.807} C_VEL
LIN {X 0,Y 39.035,Z 703.961,A -85,B 0,C 180,E1 -29822.694,E2 -29822.694} C_VEL
LIN {X 0,Y 42.76,Z 702.571,A -85,B 0,C 180,E1 -29831.107,E2 -29831.107} C_VEL
LIN {X 0,Y 49.631,Z 699.659,A -85,B 0,C 180,E1 -29841.156,E2 -29841.156} C_VEL
LIN {X 0,Y 57.707,Z 695.699,A -85,B 0,C 180,E1 -29848.489,E2 -29848.489} C_VEL
LIN {X 0,Y 66.438,Z 690.567,A -85,B 0,C 180,E1 -29854.05,E2 -29854.05} C_VEL
LIN {X 0,Y 75.598,Z 684.1,A -85,B 0,C 180,E1 -29858.383,E2 -29858.383} C_VEL
LIN {X 0,Y 85.053,Z 676.061,A -85,B 0,C 180,E1 -29861.854,E2 -29861.854} C_VEL
LIN {X 0,Y 93.171,Z 667.829,A -85,B 0,C 180,E1 -29864.105,E2 -29864.105} C_VEL
LIN {X 0,Y 101.415,Z 657.657,A -85,B 0,C 180,E1 -29865.98,E2 -29865.98} C_VEL
LIN {X 0,Y 108.917,Z 646.208,A -85,B 0,C 180,E1 -29867.416,E2 -29867.416} C_VEL
LIN {X 0,Y 114.774,Z 634.822,A -85,B 0,C 180,E1 -29868.45,E2 -29868.45} C_VEL
LIN {X 0,Y 119.41,Z 623.096,A -85,B 0,C 180,E1 -29869.165,E2 -29869.165} C_VEL
LIN {X 0,Y 123.182,Z 609.798,A -85,B 0,C 180,E1 -29869.718,E2 -29869.718} C_VEL
LIN {X 0,Y 125.527,Z 595.818,A -85,B 0,C 180,E1 -29870.077,E2 -29870.077} C_VEL
LIN {X 0,Y 129.612,Z 560.304,A -85,B 0,C 180,E1 -29870.991,E2 -29870.991} C_VEL
LIN {X 0,Y 129.138,Z 557.322,A -85,B 0,C 180,E1 -29873.751,E2 -29873.751} C_VEL
LIN {X 0,Y 128.835,Z 555.03,A -85,B 0,C 180,E1 -29876.873,E2 -29876.873} C_VEL
LIN {X 0,Y 128.795,Z 553.719,A -85,B 0,C 180,E1 -29880,E2 -29880} C_VEL
LIN {X 0,Y 129.055,Z 553.709,A -85,B 0,C 180,E1 -29883.708,E2 -29883.708} C_VEL
LIN {X 0,Y 130.017,Z 556.055,A -85,B 0,C 180,E1 -29888.814,E2 -29888.814} C_VEL
LIN {X 0,Y 129.607,Z 559.893,A -85,B 0,C 180,E1 -29889.004,E2 -29889.004} C_VEL
LIN {X 0,Y 124.367,Z 603.54,A -85,B 0,C 180,E1 -29890.058,E2 -29890.058} C_VEL
LIN {X 0,Y 121.488,Z 616.359,A -85,B 0,C 180,E1 -29890.437,E2 -29890.437} C_VEL
LIN {X 0,Y 117.249,Z 628.984,A -85,B 0,C 180,E1 -29891.025,E2 -29891.025} C_VEL
LIN {X 0,Y 112.196,Z 640.271,A -85,B 0,C 180,E1 -29891.827,E2 -29891.827} C_VEL
LIN {X 0,Y 105.49,Z 651.891,A -85,B 0,C 180,E1 -29893.001,E2 -29893.001} C_VEL
LIN {X 0,Y 98.008,Z 662.283,A -85,B 0,C 180,E1 -29894.515,E2 -29894.515} C_VEL
LIN {X 0,Y 89.784,Z 671.659,A -85,B 0,C 180,E1 -29896.483,E2 -29896.483} C_VEL
LIN {X 0,Y 80.108,Z 680.663,A -85,B 0,C 180,E1 -29899.417,E2 -29899.417} C_VEL
LIN {X 0,Y 70.729,Z 687.909,A -85,B 0,C 180,E1 -29903.199,E2 -29903.199} C_VEL
LIN {X 0,Y 63.267,Z 692.816,A -85,B 0,C 180,E1 -29907.289,E2 -29907.289} C_VEL
LIN {X 0,Y 54.694,Z 697.561,A -85,B 0,C 180,E1 -29913.358,E2 -29913.358} C_VEL
LIN {X 0,Y 46.931,Z 701.183,A -85,B 0,C 180,E1 -29921.515,E2 -29921.515} C_VEL
LIN {X 0,Y 42.494,Z 703.05,A -85,B 0,C 180,E1 -29928.579,E2 -29928.579} C_VEL
LIN {X 0,Y 38.834,Z 704.454,A -85,B 0,C 180,E1 -29937.115,E2 -29937.115} C_VEL
LIN {X 0,Y 34.568,Z 706.053,A -85,B 0,C 180,E1 -29958.268,E2 -29958.268} C_VEL
LIN {X 0,Y 34.253,Z 706.264,A -85,B 0,C 180,E1 -29969.998,E2 -29969.998} C_VEL
LIN {X 0,Y 34.57,Z 706.033,A -85,B 0,C 180,E1 -29981.728,E2 -29981.728} C_VEL
LIN {X 0,Y 36.142,Z 705.413,A -85,B 0,C 180,E1 -29992.885,E2 -29992.885} C_VEL
LIN {X 0,Y 38.834,Z 704.406,A -85,B 0,C 180,E1 -30002.882,E2 -30002.882} C_VEL
LIN {X 0,Y 42.495,Z 702.975,A -85,B 0,C 180,E1 -30011.415,E2 -30011.415} C_VEL
LIN {X 0,Y 49.422,Z 700.013,A -85,B 0,C 180,E1 -30021.454,E2 -30021.454} C_VEL
LIN {X 0,Y 57.448,Z 695.995,A -85,B 0,C 180,E1 -30028.909,E2 -30028.909} C_VEL
LIN {X 0,Y 67.697,Z 689.817,A -85,B 0,C 180,E1 -30035.242,E2 -30035.242} C_VEL
LIN {X 0,Y 77.129,Z 682.905,A -85,B 0,C 180,E1 -30039.517,E2 -30039.517} C_VEL
LIN {X 0,Y 77.82,Z 681.612,A -85,B 0,C 180,E1 -30041.911,E2 -30041.911} C_VEL
LIN {X 0,Y 78.628,Z 678.104,A -85,B 0,C 180,E1 -30054.872,E2 -30054.872} C_VEL
LIN {X 0,Y 83.41,Z 673.87,A -85,B 0,C 180,E1 -30064.834,E2 -30064.834} C_VEL
LIN {X 0,Y 92.553,Z 667.601,A -85,B 0,C 180,E1 -30074.807,E2 -30074.807} C_VEL
LIN {X 0,Y 93.179,Z 667.227,A -85,B 0,C 180,E1 -30075.414,E2 -30075.414} C_VEL
LIN {X 0,Y 91.582,Z 669.218,A -85,B 0,C 180,E1 -30076.415,E2 -30076.415} C_VEL
LIN {X 0,Y 83.495,Z 677.228,A -85,B 0,C 180,E1 -30078.748,E2 -30078.748} C_VEL
LIN {X 0,Y 74.488,Z 684.758,A -85,B 0,C 180,E1 -30082.173,E2 -30082.173} C_VEL
LIN {X 0,Y 66.462,Z 690.367,A -85,B 0,C 180,E1 -30085.996,E2 -30085.996} C_VEL
LIN {X 0,Y 57.738,Z 695.538,A -85,B 0,C 180,E1 -30091.566,E2 -30091.566} C_VEL
LIN {X 0,Y 49.541,Z 699.601,A -85,B 0,C 180,E1 -30099.101,E2 -30099.101} C_VEL
LIN {X 0,Y 45.175,Z 701.319,A -85,B 0,C 180,E1 -30103.512,E2 -30103.512} C_VEL
LIN {X 0,Y 37.27,Z 703.523,A -85,B 0,C 180,E1 -30111.311,E2 -30111.311} C_VEL
LIN {X 0,Y 31.471,Z 704.77,A -85,B 0,C 180,E1 -30120.193,E2 -30120.193} C_VEL
LIN {X 0,Y 28.428,Z 705.383,A -85,B 0,C 180,E1 -30129.864,E2 -30129.864} C_VEL
LIN {X 0,Y 27.852,Z 705.5,A -85,B 0,C 180,E1 -30133.691,E2 -30133.691} C_VEL
LIN {X 0,Y 27.082,Z 705.796,A -85,B 0,C 180,E1 -30150.002,E2 -30150.002} C_VEL
LIN {X 0,Y 27.681,Z 705.593,A -85,B 0,C 180,E1 -30164.71,E2 -30164.71} C_VEL
LIN {X 0,Y 29.85,Z 704.996,A -85,B 0,C 180,E1 -30178.095,E2 -30178.095} C_VEL
LIN {X 0,Y 33.28,Z 704.014,A -85,B 0,C 180,E1 -30189.313,E2 -30189.313} C_VEL
LIN {X 0,Y 37.684,Z 702.624,A -85,B 0,C 180,E1 -30198.247,E2 -30198.247} C_VEL
LIN {X 0,Y 45.505,Z 699.711,A -85,B 0,C 180,E1 -30208.154,E2 -30208.154} C_VEL
LIN {X 0,Y 54.326,Z 695.75,A -85,B 0,C 180,E1 -30214.904,E2 -30214.904} C_VEL
LIN {X 0,Y 63.653,Z 690.617,A -85,B 0,C 180,E1 -30219.805,E2 -30219.805} C_VEL
LIN {X 0,Y 73.275,Z 684.149,A -85,B 0,C 180,E1 -30223.566,E2 -30223.566} C_VEL
LIN {X 0,Y 83.116,Z 676.108,A -85,B 0,C 180,E1 -30226.511,E2 -30226.511} C_VEL
LIN {X 0,Y 91.483,Z 667.874,A -85,B 0,C 180,E1 -30228.383,E2 -30228.383} C_VEL
LIN {X 0,Y 99.931,Z 657.698,A -85,B 0,C 180,E1 -30229.936,E2 -30229.936} C_VEL
LIN {X 0,Y 107.592,Z 646.244,A -85,B 0,C 180,E1 -30231.113,E2 -30231.113} C_VEL
LIN {X 0,Y 113.568,Z 634.85,A -85,B 0,C 180,E1 -30231.953,E2 -30231.953} C_VEL
LIN {X 0,Y 118.712,Z 621.861,A -85,B 0,C 180,E1 -30232.589,E2 -30232.589} C_VEL
LIN {X 0,Y 122.181,Z 609.515,A -85,B 0,C 180,E1 -30232.996,E2 -30232.996} C_VEL
LIN {X 0,Y 124.5,Z 595.759,A -85,B 0,C 180,E1 -30233.291,E2 -30233.291} C_VEL
LIN {X 0,Y 128.177,Z 564.666,A -85,B 0,C 180,E1 -30233.97,E2 -30233.97} C_VEL
LIN {X 0,Y 127.907,Z 561.811,A -85,B 0,C 180,E1 -30237.736,E2 -30237.736} C_VEL
LIN {X 0,Y 127.921,Z 560.834,A -85,B 0,C 180,E1 -30240,E2 -30240} C_VEL
LIN {X 0,Y 128.182,Z 560.833,A -85,B 0,C 180,E1 -30243.733,E2 -30243.733} C_VEL
LIN {X 0,Y 128.478,Z 561.726,A -85,B 0,C 180,E1 -30245.916,E2 -30245.916} C_VEL
LIN {X 0,Y 123.317,Z 603.637,A -85,B 0,C 180,E1 -30246.813,E2 -30246.813} C_VEL
LIN {X 0,Y 120.406,Z 616.352,A -85,B 0,C 180,E1 -30247.12,E2 -30247.12} C_VEL
LIN {X 0,Y 116.103,Z 628.961,A -85,B 0,C 180,E1 -30247.592,E2 -30247.592} C_VEL
LIN {X 0,Y 110.958,Z 640.24,A -85,B 0,C 180,E1 -30248.235,E2 -30248.235} C_VEL
LIN {X 0,Y 104.125,Z 651.852,A -85,B 0,C 180,E1 -30249.198,E2 -30249.198} C_VEL
LIN {X 0,Y 96.472,Z 662.24,A -85,B 0,C 180,E1 -30250.425,E2 -30250.425} C_VEL
LIN {X 0,Y 88.034,Z 671.614,A -85,B 0,C 180,E1 -30252.049,E2 -30252.049} C_VEL
LIN {X 0,Y 78.029,Z 680.615,A -85,B 0,C 180,E1 -30254.474,E2 -30254.474} C_VEL
LIN {X 0,Y 68.239,Z 687.858,A -85,B 0,C 180,E1 -30257.695,E2 -30257.695} C_VEL
LIN {X 0,Y 60.339,Z 692.765,A -85,B 0,C 180,E1 -30261.279,E2 -30261.279} C_VEL
LIN {X 0,Y 51.127,Z 697.509,A -85,B 0,C 180,E1 -30266.681,E2 -30266.681} C_VEL
LIN {X 0,Y 42.553,Z 701.13,A -85,B 0,C 180,E1 -30274.328,E2 -30274.328} C_VEL
LIN {X 0,Y 37.44,Z 702.997,A -85,B 0,C 180,E1 -30281.332,E2 -30281.332} C_VEL
LIN {X 0,Y 33.071,Z 704.4,A -85,B 0,C 180,E1 -30290.389,E2 -30290.389} C_VEL
LIN {X 0,Y 27.652,Z 705.999,A -85,B 0,C 180,E1 -30315.274,E2 -30315.274} C_VEL
LIN {X 0,Y 27.142,Z 706.21,A -85,B 0,C 180,E1 -30329.998,E2 -30329.998} C_VEL
LIN {X 0,Y 27.655,Z 705.978,A -85,B 0,C 180,E1 -30344.72,E2 -30344.72} C_VEL
LIN {X 0,Y 29.709,Z 705.359,A -85,B 0,C 180,E1 -30358.235,E2 -30358.235} C_VEL
LIN {X 0,Y 33.071,Z 704.352,A -85,B 0,C 180,E1 -30369.607,E2 -30369.607} C_VEL
LIN {X 0,Y 37.441,Z 702.92,A -85,B 0,C 180,E1 -30378.661,E2 -30378.661} C_VEL
LIN {X 0,Y 45.335,Z 699.958,A -85,B 0,C 180,E1 -30388.497,E2 -30388.497} C_VEL
LIN {X 0,Y 54.114,Z 695.94,A -85,B 0,C 180,E1 -30395.383,E2 -30395.383} C_VEL
LIN {X 0,Y 64.201,Z 690.284,A -85,B 0,C 180,E1 -30400.601,E2 -30400.601} C_VEL
LIN {X 0,Y 69.864,Z 686.561,A -85,B 0,C 180,E1 -30402.872,E2 -30402.872} C_VEL
LIN {X 0,Y 71.693,Z 685.02,A -85,B 0,C 180,E1 -30404.573,E2 -30404.573} C_VEL
LIN {X 0,Y 72.645,Z 682.721,A -85,B 0,C 180,E1 -30414.449,E2 -30414.449} C_VEL
LIN {X 0,Y 77.682,Z 678.83,A -85,B 0,C 180,E1 -30425.632,E2 -30425.632} C_VEL
LIN {X 0,Y 83.718,Z 675.09,A -85,B 0,C 180,E1 -30432.655,E2 -30432.655} C_VEL
LIN {X 0,Y 83.141,Z 675.818,A -85,B 0,C 180,E1 -30433.566,E2 -30433.566} C_VEL
LIN {X 0,Y 73.302,Z 683.913,A -85,B 0,C 180,E1 -30436.51,E2 -30436.51} C_VEL
LIN {X 0,Y 63.672,Z 690.421,A -85,B 0,C 180,E1 -30440.248,E2 -30440.248} C_VEL
LIN {X 0,Y 54.359,Z 695.592,A -85,B 0,C 180,E1 -30445.177,E2 -30445.177} C_VEL
LIN {X 0,Y 44.923,Z 699.833,A -85,B 0,C 180,E1 -30452.548,E2 -30452.548} C_VEL
LIN {X 0,Y 37.739,Z 702.537,A -85,B 0,C 180,E1 -30461.851,E2 -30461.851} C_VEL
LIN {X 0,Y 33.323,Z 703.959,A -85,B 0,C 180,E1 -30470.751,E2 -30470.751} C_VEL
LIN {X 0,Y 27.852,Z 705.5,A -85,B 0,C 180,E1 -30493.691,E2 -30493.691} C_VEL
LIN {X 0,Y 26.338,Z 705.849,A -85,B 0,C 180,E1 -30505.735,E2 -30505.735} C_VEL
LIN {X 0,Y 24.916,Z 705.884,A -85,B 0,C 180,E1 -30518.68,E2 -30518.68} C_VEL
LIN {X 0,Y 25.204,Z 705.026,A -85,B 0,C 180,E1 -30546.402,E2 -30546.402} C_VEL
LIN {X 0,Y 27.923,Z 704.13,A -85,B 0,C 180,E1 -30557.813,E2 -30557.813} C_VEL
LIN {X 0,Y 29.229,Z 703.761,A -85,B 0,C 180,E1 -30560.76,E2 -30560.76} C_VEL
LIN {X 0,Y 33.37,Z 702.677,A -85,B 0,C 180,E1 -30567.402,E2 -30567.402} C_VEL
LIN {X 0,Y 42.186,Z 699.764,A -85,B 0,C 180,E1 -30576.392,E2 -30576.392} C_VEL
LIN {X 0,Y 51.71,Z 695.802,A -85,B 0,C 180,E1 -30582.066,E2 -30582.066} C_VEL
LIN {X 0,Y 61.563,Z 690.668,A -85,B 0,C 180,E1 -30586.019,E2 -30586.019} C_VEL
LIN {X 0,Y 71.587,Z 684.198,A -85,B 0,C 180,E1 -30589.04,E2 -30589.04} C_VEL
LIN {X 0,Y 81.749,Z 676.156,A -85,B 0,C 180,E1 -30591.369,E2 -30591.369} C_VEL
LIN {X 0,Y 90.321,Z 667.919,A -85,B 0,C 180,E1 -30592.798,E2 -30592.798} C_VEL
LIN {X 0,Y 98.937,Z 657.739,A -85,B 0,C 180,E1 -30593.989,E2 -30593.989} C_VEL
LIN {X 0,Y 106.726,Z 646.281,A -85,B 0,C 180,E1 -30594.882,E2 -30594.882} C_VEL
LIN {X 0,Y 112.794,Z 634.878,A -85,B 0,C 180,E1 -30595.523,E2 -30595.523} C_VEL
LIN {X 0,Y 118.007,Z 621.877,A -85,B 0,C 180,E1 -30596.005,E2 -30596.005} C_VEL
LIN {X 0,Y 121.564,Z 609.304,A -85,B 0,C 180,E1 -30596.324,E2 -30596.324} C_VEL
LIN {X 0,Y 124.006,Z 594.595,A -85,B 0,C 180,E1 -30596.568,E2 -30596.568} C_VEL
LIN {X 0,Y 127.026,Z 569.544,A -85,B 0,C 180,E1 -30597.065,E2 -30597.065} C_VEL
LIN {X 0,Y 127.043,Z 567.977,A -85,B 0,C 180,E1 -30600,E2 -30600} C_VEL
LIN {X 0,Y 127.221,Z 567.712,A -85,B 0,C 180,E1 -30602.81,E2 -30602.81} C_VEL
LIN {X 0,Y 122.59,Z 604.196,A -85,B 0,C 180,E1 -30603.531,E2 -30603.531} C_VEL
LIN {X 0,Y 119.516,Z 617.071,A -85,B 0,C 180,E1 -30603.763,E2 -30603.763} C_VEL
LIN {X 0,Y 114.944,Z 630.029,A -85,B 0,C 180,E1 -30604.125,E2 -30604.125} C_VEL
LIN {X 0,Y 109.297,Z 641.818,A -85,B 0,C 180,E1 -30604.661,E2 -30604.661} C_VEL
LIN {X 0,Y 102.361,Z 653.078,A -85,B 0,C 180,E1 -30605.394,E2 -30605.394} C_VEL
LIN {X 0,Y 94.58,Z 663.248,A -85,B 0,C 180,E1 -30606.344,E2 -30606.344} C_VEL
LIN {X 0,Y 86.828,Z 671.568,A -85,B 0,C 180,E1 -30607.45,E2 -30607.45} C_VEL
LIN {X 0,Y 76.563,Z 680.566,A -85,B 0,C 180,E1 -30609.318,E2 -30609.318} C_VEL
LIN {X 0,Y 66.422,Z 687.808,A -85,B 0,C 180,E1 -30611.832,E2 -30611.832} C_VEL
LIN {X 0,Y 58.131,Z 692.714,A -85,B 0,C 180,E1 -30614.713,E2 -30614.713} C_VEL
LIN {X 0,Y 48.347,Z 697.457,A -85,B 0,C 180,E1 -30619.108,E2 -30619.108} C_VEL
LIN {X 0,Y 38.99,Z 701.077,A -85,B 0,C 180,E1 -30625.672,E2 -30625.672} C_VEL
LIN {X 0,Y 33.163,Z 702.943,A -85,B 0,C 180,E1 -30632.034,E2 -30632.034} C_VEL
LIN {X 0,Y 27.953,Z 704.346,A -85,B 0,C 180,E1 -30641.035,E2 -30641.035} C_VEL
LIN {X 0,Y 23.677,Z 705.34,A -85,B 0,C 180,E1 -30653.581,E2 -30653.581} C_VEL
LIN {X 0,Y 20.847,Z 705.945,A -85,B 0,C 180,E1 -30670.295,E2 -30670.295} C_VEL
LIN {X 0,Y 20.037,Z 706.156,A -85,B 0,C 180,E1 -30689.997,E2 -30689.997} C_VEL
LIN {X 0,Y 20.849,Z 705.924,A -85,B 0,C 180,E1 -30709.697,E2 -30709.697} C_VEL
LIN {X 0,Y 23.683,Z 705.304,A -85,B 0,C 180,E1 -30726.403,E2 -30726.403} C_VEL
LIN {X 0,Y 27.953,Z 704.297,A -85,B 0,C 180,E1 -30738.959,E2 -30738.959} C_VEL
LIN {X 0,Y 33.163,Z 702.865,A -85,B 0,C 180,E1 -30747.958,E2 -30747.958} C_VEL
LIN {X 0,Y 42.05,Z 699.904,A -85,B 0,C 180,E1 -30756.814,E2 -30756.814} C_VEL
LIN {X 0,Y 51.556,Z 695.886,A -85,B 0,C 180,E1 -30762.593,E2 -30762.593} C_VEL
LIN {X 0,Y 61.334,Z 690.748,A -85,B 0,C 180,E1 -30766.521,E2 -30766.521} C_VEL
LIN {X 0,Y 64.756,Z 688.699,A -85,B 0,C 180,E1 -30767.626,E2 -30767.626} C_VEL
LIN {X 0,Y 66.477,Z 686.874,A -85,B 0,C 180,E1 -30773.932,E2 -30773.932} C_VEL
LIN {X 0,Y 71.164,Z 683.646,A -85,B 0,C 180,E1 -30785.668,E2 -30785.668} C_VEL
LIN {X 0,Y 73.56,Z 682.361,A -85,B 0,C 180,E1 -30789.175,E2 -30789.175} C_VEL
LIN {X 0,Y 71.605,Z 683.967,A -85,B 0,C 180,E1 -30791.042,E2 -30791.042} C_VEL
LIN {X 0,Y 61.578,Z 690.475,A -85,B 0,C 180,E1 -30794.043,E2 -30794.043} C_VEL
LIN {X 0,Y 51.733,Z 695.646,A -85,B 0,C 180,E1 -30798.022,E2 -30798.022} C_VEL
LIN {X 0,Y 42.218,Z 699.647,A -85,B 0,C 180,E1 -30803.713,E2 -30803.713} C_VEL
LIN {X 0,Y 33.411,Z 702.592,A -85,B 0,C 180,E1 -30812.714,E2 -30812.714} C_VEL
LIN {X 0,Y 28.185,Z 704.013,A -85,B 0,C 180,E1 -30821.58,E2 -30821.58} C_VEL
LIN {X 0,Y 20.909,Z 705.624,A -85,B 0,C 180,E1 -30850.361,E2 -30850.361} C_VEL
LIN {X 0,Y 19.992,Z 705.85,A -85,B 0,C 180,E1 -30870.003,E2 -30870.003} C_VEL
LIN {X 0,Y 20.904,Z 705.647,A -85,B 0,C 180,E1 -30889.649,E2 -30889.649} C_VEL
LIN {X 0,Y 28.14,Z 704.068,A -85,B 0,C 180,E1 -30918.53,E2 -30918.53} C_VEL
LIN {X 0,Y 29.229,Z 703.761,A -85,B 0,C 180,E1 -30920.76,E2 -30920.76} C_VEL
LIN {X 0,Y 33.164,Z 702.637,A -85,B 0,C 180,E1 -30928.571,E2 -30928.571} C_VEL
LIN {X 0,Y 39.581,Z 700.239,A -85,B 0,C 180,E1 -30939.96,E2 -30939.96} C_VEL
LIN {X 0,Y 46.891,Z 697.219,A -85,B 0,C 180,E1 -30947.928,E2 -30947.928} C_VEL
LIN {X 0,Y 51.889,Z 694.959,A -85,B 0,C 180,E1 -30950.493,E2 -30950.493} C_VEL
LIN {X 0,Y 63.682,Z 688.728,A -85,B 0,C 180,E1 -30953.35,E2 -30953.35} C_VEL
LIN {X 0,Y 74.041,Z 681.775,A -85,B 0,C 180,E1 -30955.327,E2 -30955.327} C_VEL
LIN {X 0,Y 84.475,Z 673.082,A -85,B 0,C 180,E1 -30956.733,E2 -30956.733} C_VEL
LIN {X 0,Y 93.202,Z 664.156,A -85,B 0,C 180,E1 -30957.637,E2 -30957.637} C_VEL
LIN {X 0,Y 101.075,Z 654.272,A -85,B 0,C 180,E1 -30958.273,E2 -30958.273} C_VEL
LIN {X 0,Y 108.079,Z 643.308,A -85,B 0,C 180,E1 -30958.835,E2 -30958.835} C_VEL
LIN {X 0,Y 114.217,Z 631.046,A -85,B 0,C 180,E1 -30959.242,E2 -30959.242} C_VEL
LIN {X 0,Y 118.823,Z 618.513,A -85,B 0,C 180,E1 -30959.528,E2 -30959.528} C_VEL
LIN {X 0,Y 122.195,Z 605.045,A -85,B 0,C 180,E1 -30959.732,E2 -30959.732} C_VEL
LIN {X 0,Y 124.517,Z 588.547,A -85,B 0,C 180,E1 -30959.944,E2 -30959.944} C_VEL
LIN {X 0,Y 122.03,Z 605.835,A -85,B 0,C 180,E1 -30960.229,E2 -30960.229} C_VEL
LIN {X 0,Y 118.602,Z 619.242,A -85,B 0,C 180,E1 -30960.416,E2 -30960.416} C_VEL
LIN {X 0,Y 114.213,Z 631.056,A -85,B 0,C 180,E1 -30960.603,E2 -30960.603} C_VEL
LIN {X 0,Y 108.073,Z 643.328,A -85,B 0,C 180,E1 -30960.99,E2 -30960.99} C_VEL
LIN {X 0,Y 101.063,Z 654.304,A -85,B 0,C 180,E1 -30961.481,E2 -30961.481} C_VEL
LIN {X 0,Y 93.186,Z 664.202,A -85,B 0,C 180,E1 -30962.116,E2 -30962.116} C_VEL
LIN {X 0,Y 84.449,Z 673.142,A -85,B 0,C 180,E1 -30962.939,E2 -30962.939} C_VEL
LIN {X 0,Y 73.998,Z 681.853,A -85,B 0,C 180,E1 -30964.24,E2 -30964.24} C_VEL
LIN {X 0,Y 63.608,Z 688.828,A -85,B 0,C 180,E1 -30966.051,E2 -30966.051} C_VEL
LIN {X 0,Y 53.315,Z 694.383,A -85,B 0,C 180,E1 -30968.633,E2 -30968.633} C_VEL
LIN {X 0,Y 43.136,Z 698.733,A -85,B 0,C 180,E1 -30972.154,E2 -30972.154} C_VEL
LIN {X 0,Y 36.478,Z 701.024,A -85,B 0,C 180,E1 -30975.559,E2 -30975.559} C_VEL
LIN {X 0,Y 29.995,Z 702.89,A -85,B 0,C 180,E1 -30980.403,E2 -30980.403} C_VEL
LIN {X 0,Y 23.891,Z 704.293,A -85,B 0,C 180,E1 -30988.047,E2 -30988.047} C_VEL
LIN {X 0,Y 14.359,Z 705.892,A -85,B 0,C 180,E1 -31020.692,E2 -31020.692} C_VEL
LIN {X 0,Y 12.945,Z 706.102,A -85,B 0,C 180,E1 -31049.996,E2 -31049.996} C_VEL
LIN {X 0,Y 14.361,Z 705.87,A -85,B 0,C 180,E1 -31079.295,E2 -31079.295} C_VEL
LIN {X 0,Y 23.89,Z 704.243,A -85,B 0,C 180,E1 -31111.947,E2 -31111.947} C_VEL
LIN {X 0,Y 29.995,Z 702.811,A -85,B 0,C 180,E1 -31119.587,E2 -31119.587} C_VEL
LIN {X 0,Y 39.787,Z 699.849,A -85,B 0,C 180,E1 -31126.287,E2 -31126.287} C_VEL
LIN {X 0,Y 49.892,Z 695.832,A -85,B 0,C 180,E1 -31130.411,E2 -31130.411} C_VEL
LIN {X 0,Y 56.735,Z 692.497,A -85,B 0,C 180,E1 -31132.3,E2 -31132.3} C_VEL
LIN {X 0,Y 59.71,Z 690.892,A -85,B 0,C 180,E1 -31133.241,E2 -31133.241} C_VEL
LIN {X 0,Y 64.723,Z 687.875,A -85,B 0,C 180,E1 -31146.234,E2 -31146.234} C_VEL
LIN {X 0,Y 63.695,Z 688.538,A -85,B 0,C 180,E1 -31146.762,E2 -31146.762} C_VEL
LIN {X 0,Y 53.388,Z 694.109,A -85,B 0,C 180,E1 -31149.146,E2 -31149.146} C_VEL
LIN {X 0,Y 43.231,Z 698.477,A -85,B 0,C 180,E1 -31152.735,E2 -31152.735} C_VEL
LIN {X 0,Y 36.582,Z 700.775,A -85,B 0,C 180,E1 -31156.143,E2 -31156.143} C_VEL
LIN {X 0,Y 30.157,Z 702.647,A -85,B 0,C 180,E1 -31161.228,E2 -31161.228} C_VEL
LIN {X 0,Y 24.061,Z 704.068,A -85,B 0,C 180,E1 -31168.807,E2 -31168.807} C_VEL
LIN {X 0,Y 14.415,Z 705.678,A -85,B 0,C 180,E1 -31200.825,E2 -31200.825} C_VEL
LIN {X 0,Y 12.912,Z 705.904,A -85,B 0,C 180,E1 -31230.004,E2 -31230.004} C_VEL
LIN {X 0,Y 14.411,Z 705.701,A -85,B 0,C 180,E1 -31259.194,E2 -31259.194} C_VEL
LIN {X 0,Y 24.021,Z 704.122,A -85,B 0,C 180,E1 -31291.377,E2 -31291.377} C_VEL
LIN {X 0,Y 30.131,Z 702.731,A -85,B 0,C 180,E1 -31298.913,E2 -31298.913} C_VEL
LIN {X 0,Y 39.874,Z 699.816,A -85,B 0,C 180,E1 -31305.797,E2 -31305.797} C_VEL
LIN {X 0,Y 51.889,Z 694.959,A -85,B 0,C 180,E1 -31310.493,E2 -31310.493} C_VEL
LIN {X 0,Y 51.94,Z 694.884,A -85,B 0,C 180,E1 -31311.445,E2 -31311.445} C_VEL
LIN {X 0,Y 50.414,Z 695.478,A -85,B 0,C 180,E1 -31313.389,E2 -31313.389} C_VEL
LIN {X 0,Y 46.392,Z 697.105,A -85,B 0,C 180,E1 -31316.167,E2 -31316.167} C_VEL
LIN {X 0,Y 39.868,Z 699.466,A -85,B 0,C 180,E1 -31319.431,E2 -31319.431} C_VEL
LIN {X 0,Y 34.743,Z 701.09,A -85,B 0,C 180,E1 -31322.334,E2 -31322.334} C_VEL
LIN {X 0,Y 26.924,Z 703.141,A -85,B 0,C 180,E1 -31327.247,E2 -31327.247} C_VEL
LIN {X 0,Y 24.261,Z 703.664,A -85,B 0,C 180,E1 -31328.971,E2 -31328.971} C_VEL
LIN {X 0,Y 14.853,Z 705.232,A -85,B 0,C 180,E1 -31338.847,E2 -31338.847} C_VEL
LIN {X 0,Y 8.864,Z 705.837,A -85,B 0,C 180,E1 -31357.538,E2 -31357.538} C_VEL
LIN {X 0,Y 5.842,Z 706.047,A -85,B 0,C 180,E1 -31409.991,E2 -31409.991} C_VEL
LIN {X 0,Y 8.865,Z 705.815,A -85,B 0,C 180,E1 -31462.438,E2 -31462.438} C_VEL
LIN {X 0,Y 21.479,Z 704.188,A -85,B 0,C 180,E1 -31488.989,E2 -31488.989} C_VEL
LIN {X 0,Y 28.308,Z 702.756,A -85,B 0,C 180,E1 -31493.242,E2 -31493.242} C_VEL
LIN {X 0,Y 38.723,Z 699.795,A -85,B 0,C 180,E1 -31496.572,E2 -31496.572} C_VEL
LIN {X 0,Y 49.21,Z 695.778,A -85,B 0,C 180,E1 -31498.599,E2 -31498.599} C_VEL
LIN {X 0,Y 52.15,Z 694.439,A -85,B 0,C 180,E1 -31498.963,E2 -31498.963} C_VEL
LIN {X 0,Y 55.088,Z 693.017,A -85,B 0,C 180,E1 -31500,E2 -31500} C_VEL
LIN {X 0,Y 52.161,Z 694.421,A -85,B 0,C 180,E1 -31501.558,E2 -31501.558} C_VEL
LIN {X 0,Y 42.237,Z 698.532,A -85,B 0,C 180,E1 -31503.281,E2 -31503.281} C_VEL
LIN {X 0,Y 35.272,Z 700.83,A -85,B 0,C 180,E1 -31504.967,E2 -31504.967} C_VEL
LIN {X 0,Y 28.365,Z 702.702,A -85,B 0,C 180,E1 -31507.667,E2 -31507.667} C_VEL
LIN {X 0,Y 21.551,Z 704.122,A -85,B 0,C 180,E1 -31511.956,E2 -31511.956} C_VEL
LIN {X 0,Y 8.918,Z 705.732,A -85,B 0,C 180,E1 -31538.003,E2 -31538.003} C_VEL
LIN {X 0,Y 5.819,Z 705.958,A -85,B 0,C 180,E1 -31590.009,E2 -31590.009} C_VEL
LIN {X 0,Y 8.915,Z 705.755,A -85,B 0,C 180,E1 -31642.038,E2 -31642.038} C_VEL
LIN {X 0,Y 14.92,Z 705.158,A -85,B 0,C 180,E1 -31660.423,E2 -31660.423} C_VEL
LIN {X 0,Y 21.536,Z 704.175,A -85,B 0,C 180,E1 -31668.258,E2 -31668.258} C_VEL
LIN {X 0,Y 28.356,Z 702.784,A -85,B 0,C 180,E1 -31672.493,E2 -31672.493} C_VEL
LIN {X 0,Y 38.748,Z 699.869,A -85,B 0,C 180,E1 -31676.039,E2 -31676.039} C_VEL
LIN {X 0,Y 50.604,Z 695.279,A -85,B 0,C 180,E1 -31678.289,E2 -31678.289} C_VEL
LIN {X 0,Y 58.05,Z 691.674,A -85,B 0,C 180,E1 -31679.184,E2 -31679.184} C_VEL
LIN {X 0,Y 60.125,Z 690.555,A -85,B 0,C 180,E1 -31680,E2 -31680} C_VEL
LIN {X 0,Y 49.212,Z 695.927,A -85,B 0,C 180,E1 -31681.396,E2 -31681.396} C_VEL
LIN {X 0,Y 38.724,Z 699.906,A -85,B 0,C 180,E1 -31683.408,E2 -31683.408} C_VEL
LIN {X 0,Y 28.309,Z 702.837,A -85,B 0,C 180,E1 -31686.748,E2 -31686.748} C_VEL
LIN {X 0,Y 24.261,Z 703.664,A -85,B 0,C 180,E1 -31688.971,E2 -31688.971} C_VEL
LIN {X 0,Y 24.261,Z 703.664,A -85,B 0,C 180,E1 -31688.971,E2 -31688.971}

QRS_NEXT_CUT()

QRS_NEXT()
QRS_HOME()

END
